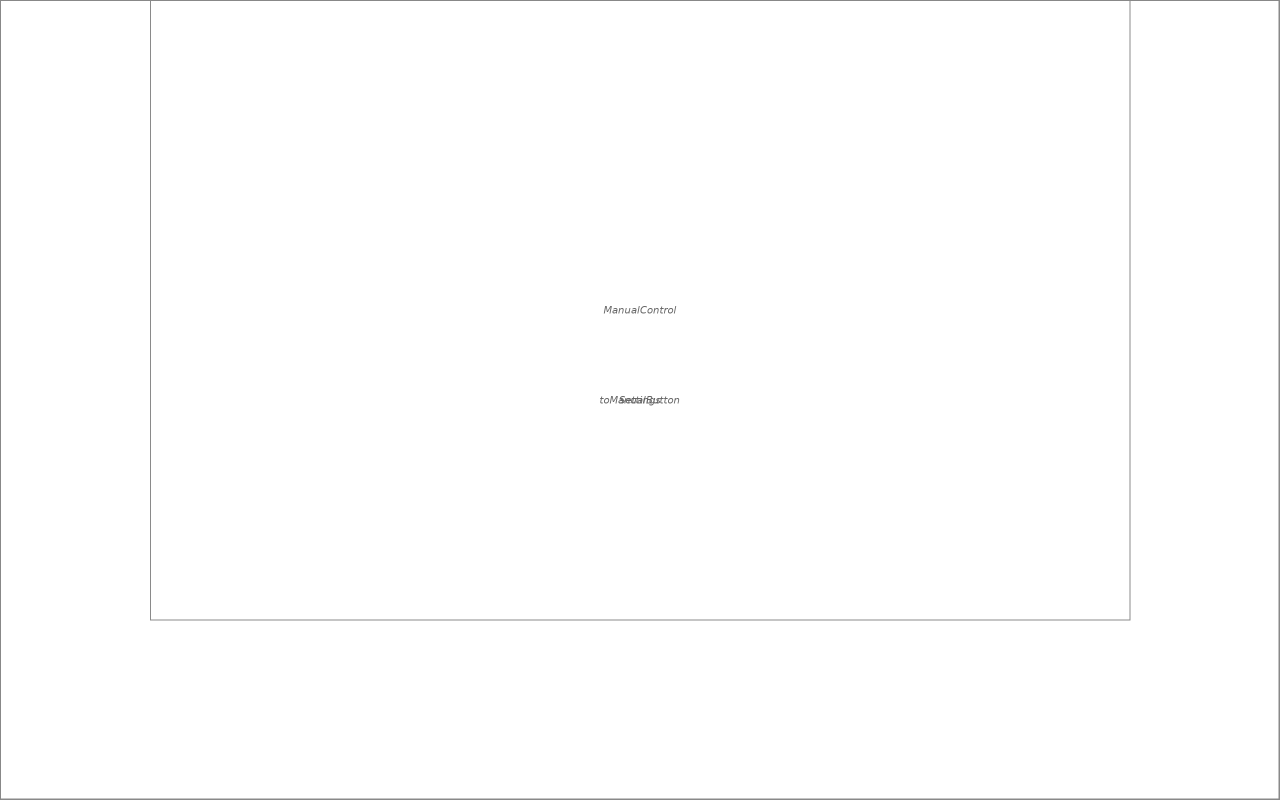
VISUALIZATION Manual  // 1280x800
VAR_IN_OUT
	bCmdParameter : BOOL ;
	nUnitsProduced : UDINT ; // Units produced in machine lifetime
END_VAR
    Frame (0,0 1280x800)
        shows toManualButton()
    Frame (0,0 1280x800)
        shows Settings(bCmdParameter := bCmdParameter, nUnitsProduced := nUnitsProduced)
    Frame (150,0 980x620)
        shows ManualControl(fbManualControler := IBF_Devices.GVL_DevManual.fbManualControler)
END_VISUALIZATION

(* stored: Version 1.1.0.1, ProductVersion 3.1.4024.9
   Visu Manual: Id {8b12630b-f7fc-46df-9948-3293bcc3e0af} *)
